Staubli VAL3: f2_place.pgx

program f2_place(mdesc x_mMdesc, mdesc x_mMdesc_slow)
  local point l_pPoint_blow
  local point l_pPoint_drop
  local point l_pPoint_safe
begin
  //vertical drop filter-2 process

  //control point preparation
  l_pPoint_safe=f2place
  l_pPoint_safe.trsf.z=l_pPoint_safe.trsf.z+nNum_safe_h

  l_pPoint_blow=f2place
  l_pPoint_blow.trsf.z=l_pPoint_blow.trsf.z+nNum_blow_h

  l_pPoint_drop=f2place

  ////to place via safe
  movej(l_pPoint_safe,t1,x_mMdesc)
  movej(l_pPoint_drop,t1,x_mMdesc)
  waitEndMove()
  //vg off
  if ioStatus(t1.gripper) >= 0
    close(t1)
  endIf
  if ioStatus(dDio_t1_vb) >= 0
    dDio_t1_vb=true
  endIf

    //on and delay
    delay(nNum_blow_delay)
    //to blow end
    movej(l_pPoint_blow,t1,x_mMdesc_slow)
    waitEndMove()
  //vb off
  if ioStatus(dDio_t1_vb) >= 0
     dDio_t1_vb=false
  endIf

    //to safe
    movej(l_pPoint_safe,t1,x_mMdesc)
    waitEndMove()
end
